// TIA Portal V19 export
VAR_GLOBAL   // PLC tag table "D27"
   D27_Lp_EntryReq_LB327 AT %Q350.6 : Bool;   // 275SH1
   D27_Lp_SafetyReset_LB327 AT %Q350.7 : Bool;   // 275SH2
   D27_Pb_EntryReq_LB327 AT %I350.6 : Bool;   // 275SH1
   D27_Pb_SafetyReset_LB327 AT %I350.7 : Bool;   // 275SH2
   D27_Ls_Os1 AT %I1500.2 : Bool;   // 350DI2 - 275A1
   D27_Ls_Os2 AT %I1500.6 : Bool;   // 350DI6 - 275A1
   D27_Comando_Elettroserratura AT %Q350.4 : Bool;   // 26202
   D27_Funzione_AUX_Elettroserratura AT %Q350.5 : Bool;   // 27505
   D27_Cancello_Chiuso AT %I350.4 : Bool;   // 27501
   D27_Cancello_Bloccato AT %I350.5 : Bool;   // 27503
END_VAR
